// TIA Portal project "Project3" (V15.1)

(* hardware
DEVICE "S71500/ET200MP station_1"  S7-1500 station
   slot 0: "Rail_0"  Rack  6ES7 590-1***0-0AA0
   slot 1: "PLC_1"  CPU 1515-2 PN  6ES7 515-2AM01-0AB0  V2.6
      slot 3: "CPU display_1"  6ES7591-1BA00-0AA0
*)

// ===== PLC "PLC_1"  CPU 1515-2 PN =====

VAR_GLOBAL   // PLC tag table "Default tag table"
   "onss1" AT %M0.0 : Bool;
   "vari" AT %M0.1 : Bool;
   "onss2" AT %M0.2 : Bool;
   "LetIEMPTY" AT %M0.3 : Bool;
   "onss3" AT %M0.4 : Bool;
   "setACTI" AT %M0.5 : Bool;
END_VAR

TYPE "CodeBar"
   STRUCT
      CodeBar : Array[0..8] of Char;
   END_STRUCT;
END_TYPE

DATA_BLOCK "AnalyseCodeBar_DB"   // DB1
{ S7_Optimized_Access := 'TRUE' }
VERSION : 0.1
// stored: InstanceOfName AnalyseCodeBar
"AnalyseCodeBar"
BEGIN
END_DATA_BLOCK

DATA_BLOCK "SysVariables"   // DB2
{ S7_Optimized_Access := 'TRUE' }
VERSION : 0.1
   VAR
      Start : Bool;
      Stop : Bool;
      SysActivated : Bool;
      SysRunning : Bool;
      ActivateSys : Bool;
      usedPPP : Int;
      usedQQ : Int;
      usedD : Int;
      WidgetsQ : Int;
      DoodadsQ : Int;
      WockiesQ : Int;
      CodeBar : String;
      InCodeBar : String;
      AcCodeBar : String;
      PrCodeBar : String;
      onss1 : Bool;
      onss2 : Bool;
      onss3 : Bool;
      onss4 : Bool;
      Oki1 : Bool;
      Oki2 : Bool;
      productType : String;
   END_VAR
BEGIN
END_DATA_BLOCK

DATA_BLOCK "DetectBarCode_DB"   // DB3
{ S7_Optimized_Access := 'TRUE' }
VERSION : 0.1
// stored: InstanceOfName DetectBarCode
"DetectBarCode"
BEGIN
END_DATA_BLOCK

FUNCTION_BLOCK "AnalyseCodeBar"   // FB1, LAD
{ S7_Optimized_Access := 'TRUE' }
VERSION : 0.1
   VAR_INPUT
      ReadedCodeBar : String;
   END_VAR
   VAR_OUTPUT
      PPPportionInt : Int;
      QQportionInt : Int;
      DportionInt : Int;
   END_VAR
   VAR
      PastCodeBar : String;
      ActuelCodeBar : String;
      UsedCodeBar : String;
      ons1 : Bool;
      ons2 : Bool;
      ons3 : Bool;
      ons4 : Bool;
      ons5 : Bool;
      PPPportion : String;
      QQportion : String;
      Dportion : String;
   END_VAR
   VAR_TEMP
      tempPPP : String;
      tempQQ : String;
      tempD : String;
   END_VAR
   VAR_TEMP   // added for the SCL form of the ladder/FBD networks
      _w1 : Bool;
      _w2 : Bool;
   END_VAR
BEGIN

REGION Network 1
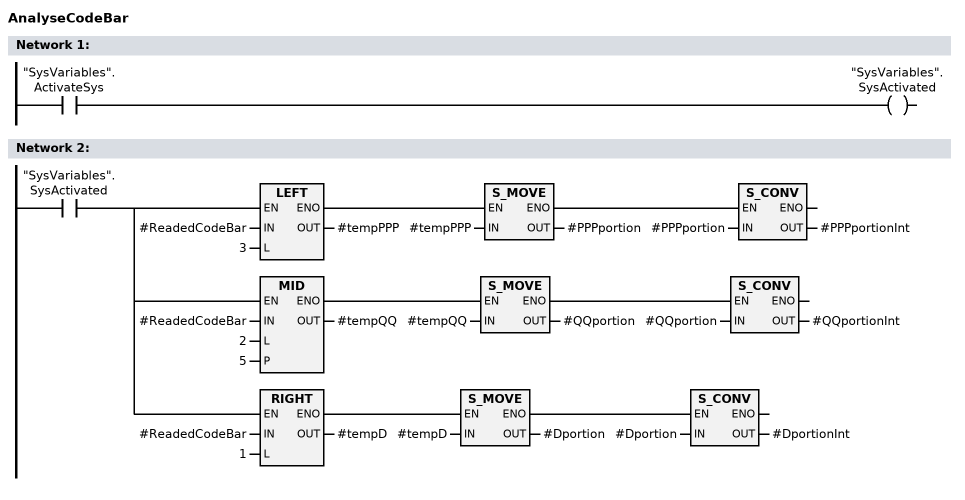
   RUNG wire#powerrail
      Contact( "SysVariables".ActivateSys )
      Coil( "SysVariables".SysActivated )
   END_RUNG
   // the same network as SCL:
   "SysVariables".SysActivated := "SysVariables".ActivateSys;
END_REGION

REGION Network 2
   #_w1 := "SysVariables".SysActivated;
   #_w2 := "SysVariables".SysActivated;
   IF #_w2 THEN
       #tempPPP := LEFT(IN := #ReadedCodeBar, L := 3);
       #PPPportion := #tempPPP;
       #PPPportionInt := S_CONV(IN := #PPPportion);
   END_IF;
   IF #_w1 THEN
       #tempQQ := MID(IN := #ReadedCodeBar, L := 2, P := 5);
       #QQportion := #tempQQ;
       #QQportionInt := S_CONV(IN := #QQportion);
       #tempD := RIGHT(IN := #ReadedCodeBar, L := 1);
       #Dportion := #tempD;
       #DportionInt := S_CONV(IN := #Dportion);
   END_IF;
END_REGION
END_FUNCTION_BLOCK

FUNCTION_BLOCK "DetectBarCode"   // FB2, LAD
{ S7_Optimized_Access := 'TRUE' }
VERSION : 0.1
   VAR_INPUT
      PPPToDetect : Int;
      QQToDetect : Int;
      DToDetect : Int;
   END_VAR
   VAR_OUTPUT
      ProductDirection : String;
      ProductType : String;
      QuanAdded : Int;
      QuanSubded : Int;
   END_VAR
   VAR_IN_OUT
      WidgetsQuan : Int;
      DoodadsQuan : Int;
      WockiesQuan : Int;
   END_VAR
   VAR
      QQPrev : Int;
      QQActuel : Int;
      ons1 : Bool;
      ons2 : Bool;
      ons3 : Bool;
      ons4 : Bool;
      ons5 : Bool;
      ons6 : Bool;
      ons7 : Bool;
      ons8 : Bool;
      ons9 : Bool;
      ons10 : Bool;
      ons11 : Bool;
      ons12 : Bool;
      ons13 : Bool;
      ons14 : Bool;
      ons15 : Bool;
      ons16 : Bool;
      ons17 : Bool;
      ons18 : Bool;
      Tap1 : Bool;
      Tap2 : Bool;
      Tap3 : Bool;
      PPPActuel : Int;
      DActuel : Int;
      PPPPrev : Int;
      DPrev : Int;
      omi1 : Bool;
   END_VAR
   VAR_TEMP
      var1 : Bool;
   END_VAR
   VAR_TEMP   // added for the SCL form of the ladder/FBD networks
      _w1 : Bool;
      _w2 : Bool;
      _w3 : Bool;
      _w4 : Bool;
      _w5 : Bool;
      _w6 : Bool;
      _w7 : Bool;
      _w8 : Bool;
      _w9 : Bool;
      _w10 : Bool;
      _w11 : Bool;
      _w12 : Bool;
      _w13 : Bool;
      _w14 : Bool;
      _w15 : Bool;
      _w16 : Bool;
      _w17 : Bool;
      _w18 : Bool;
   END_VAR
BEGIN

REGION Network 1: PPP to detect
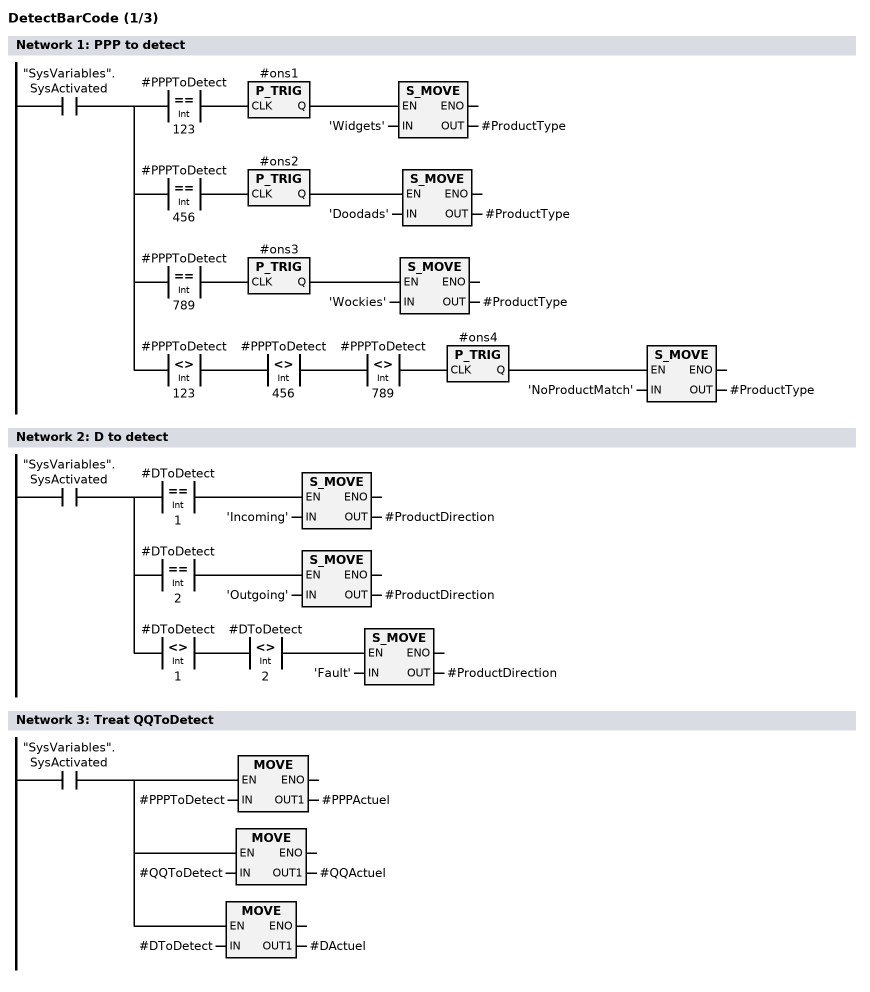
   RUNG wire#powerrail
      Contact( "SysVariables".SysActivated )
      wire#w1
      { S7_Templates := "SrcType := Int" } EQ_Contact(in1 := #PPPToDetect, in2 := 123)
      P_Trig( #ons1 )
      S_Move(in := 'Widgets', out => #ProductType)
   END_RUNG
   RUNG wire#w1
      { S7_Templates := "SrcType := Int" } EQ_Contact(in1 := #PPPToDetect, in2 := 456)
      P_Trig( #ons2 )
      S_Move(in := 'Doodads', out => #ProductType)
   END_RUNG
   RUNG wire#w1
      { S7_Templates := "SrcType := Int" } EQ_Contact(in1 := #PPPToDetect, in2 := 789)
      P_Trig( #ons3 )
      S_Move(in := 'Wockies', out => #ProductType)
   END_RUNG
   RUNG wire#w1
      { S7_Templates := "SrcType := Int" } NE_Contact(in1 := #PPPToDetect, in2 := 123)
      { S7_Templates := "SrcType := Int" } NE_Contact(in1 := #PPPToDetect, in2 := 456)
      { S7_Templates := "SrcType := Int" } NE_Contact(in1 := #PPPToDetect, in2 := 789)
      P_Trig( #ons4 )
      S_Move(in := 'NoProductMatch', out => #ProductType)
   END_RUNG
   // the same network as SCL:
   #_w1 := "SysVariables".SysActivated AND (#PPPToDetect = 123);
   #_w2 := #_w1 AND NOT #ons1;   // rising edge
   #ons1 := #_w1;
   IF #_w2 THEN #ProductType := 'Widgets'; END_IF;
   #_w3 := "SysVariables".SysActivated AND (#PPPToDetect = 456);
   #_w4 := #_w3 AND NOT #ons2;   // rising edge
   #ons2 := #_w3;
   IF #_w4 THEN #ProductType := 'Doodads'; END_IF;
   #_w5 := "SysVariables".SysActivated AND (#PPPToDetect = 789);
   #_w6 := #_w5 AND NOT #ons3;   // rising edge
   #ons3 := #_w5;
   IF #_w6 THEN #ProductType := 'Wockies'; END_IF;
   #_w7 := "SysVariables".SysActivated AND (#PPPToDetect <> 123) AND (#PPPToDetect <> 456) AND (#PPPToDetect <> 789);
   #_w8 := #_w7 AND NOT #ons4;   // rising edge
   #ons4 := #_w7;
   IF #_w8 THEN #ProductType := 'NoProductMatch'; END_IF;
END_REGION

REGION Network 2: D to detect
   RUNG wire#powerrail
      Contact( "SysVariables".SysActivated )
      wire#w1
      { S7_Templates := "SrcType := Int" } EQ_Contact(in1 := #DToDetect, in2 := 1)
      S_Move(in := 'Incoming', out => #ProductDirection)
   END_RUNG
   RUNG wire#w1
      { S7_Templates := "SrcType := Int" } EQ_Contact(in1 := #DToDetect, in2 := 2)
      S_Move(in := 'Outgoing', out => #ProductDirection)
   END_RUNG
   RUNG wire#w1
      { S7_Templates := "SrcType := Int" } NE_Contact(in1 := #DToDetect, in2 := 1)
      { S7_Templates := "SrcType := Int" } NE_Contact(in1 := #DToDetect, in2 := 2)
      S_Move(in := 'Fault', out => #ProductDirection)
   END_RUNG
   // the same network as SCL:
   IF "SysVariables".SysActivated AND (#DToDetect = 1) THEN #ProductDirection := 'Incoming'; END_IF;
   IF "SysVariables".SysActivated AND (#DToDetect = 2) THEN #ProductDirection := 'Outgoing'; END_IF;
   IF "SysVariables".SysActivated AND (#DToDetect <> 1) AND (#DToDetect <> 2) THEN
       #ProductDirection := 'Fault';
   END_IF;
END_REGION

REGION Network 3: Treat QQToDetect
   RUNG wire#powerrail
      Contact( "SysVariables".SysActivated )
      wire#w1
      Move(in := #PPPToDetect, out1 => #PPPActuel)
   END_RUNG
   RUNG wire#w1
      Move(in := #QQToDetect, out1 => #QQActuel)
   END_RUNG
   RUNG wire#w1
      Move(in := #DToDetect, out1 => #DActuel)
   END_RUNG
   // the same network as SCL:
   IF "SysVariables".SysActivated THEN
       #PPPActuel := #PPPToDetect;
       #QQActuel := #QQToDetect;
       #DActuel := #DToDetect;
   END_IF;
END_REGION

REGION Network 4: QQ to detect
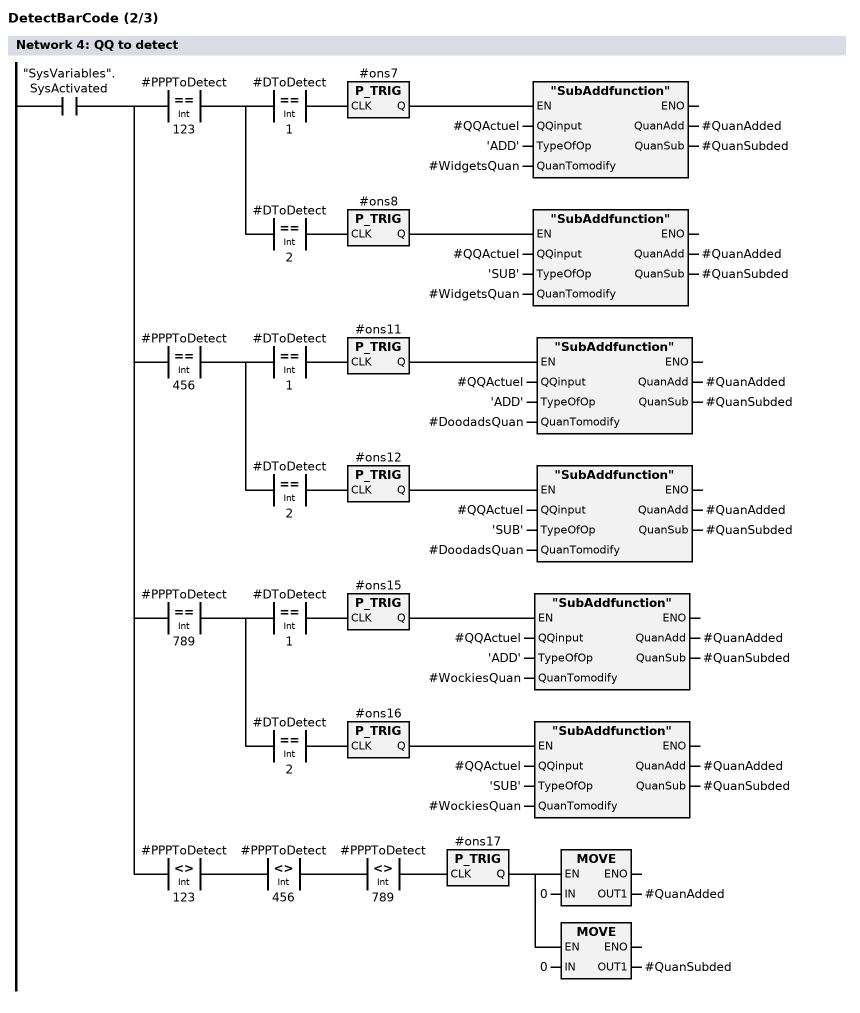
   RUNG wire#powerrail
      Contact( "SysVariables".SysActivated )
      wire#w1
      { S7_Templates := "SrcType := Int" } EQ_Contact(in1 := #PPPToDetect, in2 := 123)
      wire#w2
      { S7_Templates := "SrcType := Int" } EQ_Contact(in1 := #DToDetect, in2 := 1)
      P_Trig( #ons7 )
      "SubAddfunction"(QQinput := #QQActuel, TypeOfOp := 'ADD', QuanTomodify := #WidgetsQuan, QuanAdd => #QuanAdded, QuanSub => #QuanSubded)
   END_RUNG
   RUNG wire#w2
      { S7_Templates := "SrcType := Int" } EQ_Contact(in1 := #DToDetect, in2 := 2)
      P_Trig( #ons8 )
      "SubAddfunction"(QQinput := #QQActuel, TypeOfOp := 'SUB', QuanTomodify := #WidgetsQuan, QuanAdd => #QuanAdded, QuanSub => #QuanSubded)
   END_RUNG
   RUNG wire#w1
      { S7_Templates := "SrcType := Int" } EQ_Contact(in1 := #PPPToDetect, in2 := 456)
      wire#w3
      { S7_Templates := "SrcType := Int" } EQ_Contact(in1 := #DToDetect, in2 := 1)
      P_Trig( #ons11 )
      "SubAddfunction"(QQinput := #QQActuel, TypeOfOp := 'ADD', QuanTomodify := #DoodadsQuan, QuanAdd => #QuanAdded, QuanSub => #QuanSubded)
   END_RUNG
   RUNG wire#w3
      { S7_Templates := "SrcType := Int" } EQ_Contact(in1 := #DToDetect, in2 := 2)
      P_Trig( #ons12 )
      "SubAddfunction"(QQinput := #QQActuel, TypeOfOp := 'SUB', QuanTomodify := #DoodadsQuan, QuanAdd => #QuanAdded, QuanSub => #QuanSubded)
   END_RUNG
   RUNG wire#w1
      { S7_Templates := "SrcType := Int" } EQ_Contact(in1 := #PPPToDetect, in2 := 789)
      wire#w4
      { S7_Templates := "SrcType := Int" } EQ_Contact(in1 := #DToDetect, in2 := 1)
      P_Trig( #ons15 )
      "SubAddfunction"(QQinput := #QQActuel, TypeOfOp := 'ADD', QuanTomodify := #WockiesQuan, QuanAdd => #QuanAdded, QuanSub => #QuanSubded)
   END_RUNG
   RUNG wire#w4
      { S7_Templates := "SrcType := Int" } EQ_Contact(in1 := #DToDetect, in2 := 2)
      P_Trig( #ons16 )
      "SubAddfunction"(QQinput := #QQActuel, TypeOfOp := 'SUB', QuanTomodify := #WockiesQuan, QuanAdd => #QuanAdded, QuanSub => #QuanSubded)
   END_RUNG
   RUNG wire#w1
      { S7_Templates := "SrcType := Int" } NE_Contact(in1 := #PPPToDetect, in2 := 123)
      { S7_Templates := "SrcType := Int" } NE_Contact(in1 := #PPPToDetect, in2 := 456)
      { S7_Templates := "SrcType := Int" } NE_Contact(in1 := #PPPToDetect, in2 := 789)
      P_Trig( #ons17 )
      wire#w5
      Move(in := 0, out1 => #QuanAdded)
   END_RUNG
   RUNG wire#w5
      Move(in := 0, out1 => #QuanSubded)
   END_RUNG
   // the same network as SCL:
   #_w1 := "SysVariables".SysActivated AND (#PPPToDetect = 123);
   #_w2 := #_w1 AND (#DToDetect = 1);
   #_w3 := #_w2 AND NOT #ons7;   // rising edge
   #ons7 := #_w2;
   #_w4 := "SysVariables".SysActivated;
   IF #_w3 THEN
       "SubAddfunction"(QQinput := #QQActuel,
                        TypeOfOp := 'ADD',
                        QuanTomodify := #WidgetsQuan,
                        QuanAdd => #QuanAdded,
                        QuanSub => #QuanSubded);
   END_IF;
   #_w5 := #_w1 AND (#DToDetect = 2);
   #_w6 := #_w5 AND NOT #ons8;   // rising edge
   #ons8 := #_w5;
   IF #_w6 THEN
       "SubAddfunction"(QQinput := #QQActuel,
                        TypeOfOp := 'SUB',
                        QuanTomodify := #WidgetsQuan,
                        QuanAdd => #QuanAdded,
                        QuanSub => #QuanSubded);
   END_IF;
   #_w7 := #_w4 AND (#PPPToDetect = 456);
   #_w8 := #_w7 AND (#DToDetect = 1);
   #_w9 := #_w8 AND NOT #ons11;   // rising edge
   #ons11 := #_w8;
   IF #_w9 THEN
       "SubAddfunction"(QQinput := #QQActuel,
                        TypeOfOp := 'ADD',
                        QuanTomodify := #DoodadsQuan,
                        QuanAdd => #QuanAdded,
                        QuanSub => #QuanSubded);
   END_IF;
   #_w10 := #_w7 AND (#DToDetect = 2);
   #_w11 := #_w10 AND NOT #ons12;   // rising edge
   #ons12 := #_w10;
   IF #_w11 THEN
       "SubAddfunction"(QQinput := #QQActuel,
                        TypeOfOp := 'SUB',
                        QuanTomodify := #DoodadsQuan,
                        QuanAdd => #QuanAdded,
                        QuanSub => #QuanSubded);
   END_IF;
   #_w12 := #_w4 AND (#PPPToDetect = 789);
   #_w13 := #_w12 AND (#DToDetect = 1);
   #_w14 := #_w13 AND NOT #ons15;   // rising edge
   #ons15 := #_w13;
   IF #_w14 THEN
       "SubAddfunction"(QQinput := #QQActuel,
                        TypeOfOp := 'ADD',
                        QuanTomodify := #WockiesQuan,
                        QuanAdd => #QuanAdded,
                        QuanSub => #QuanSubded);
   END_IF;
   #_w15 := #_w12 AND (#DToDetect = 2);
   #_w16 := #_w15 AND NOT #ons16;   // rising edge
   #ons16 := #_w15;
   IF #_w16 THEN
       "SubAddfunction"(QQinput := #QQActuel,
                        TypeOfOp := 'SUB',
                        QuanTomodify := #WockiesQuan,
                        QuanAdd => #QuanAdded,
                        QuanSub => #QuanSubded);
   END_IF;
   #_w17 := #_w4 AND (#PPPToDetect <> 123) AND (#PPPToDetect <> 456) AND (#PPPToDetect <> 789);
   #_w18 := #_w17 AND NOT #ons17;   // rising edge
   #ons17 := #_w17;
   IF #_w18 THEN
       #QuanAdded := 0;
       #QuanSubded := 0;
   END_IF;
END_REGION

REGION Network 5
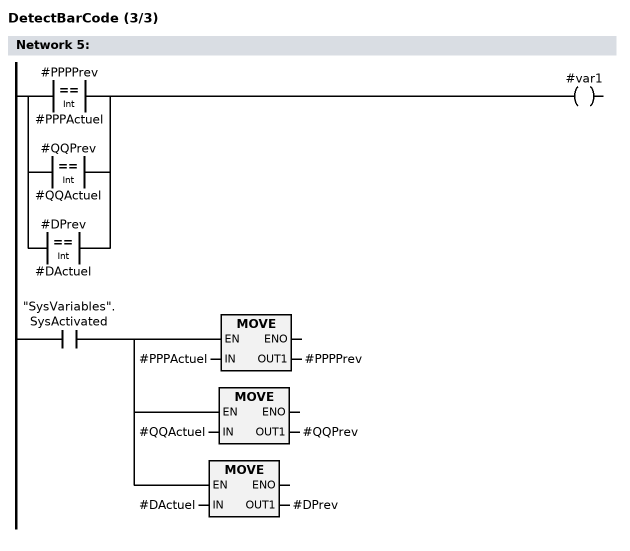
   RUNG wire#powerrail
      { S7_Templates := "SrcType := Int" } EQ_Contact(in1 := #PPPPrev, in2 := #PPPActuel)
      wire#w1
      Coil( #var1 )
   END_RUNG
   RUNG wire#powerrail
      { S7_Templates := "SrcType := Int" } EQ_Contact(in1 := #QQPrev, in2 := #QQActuel)
   END_RUNG wire#w1
   RUNG wire#powerrail
      { S7_Templates := "SrcType := Int" } EQ_Contact(in1 := #DPrev, in2 := #DActuel)
   END_RUNG wire#w1
   RUNG wire#powerrail
      Contact( "SysVariables".SysActivated )
      wire#w2
      Move(in := #PPPActuel, out1 => #PPPPrev)
   END_RUNG
   RUNG wire#w2
      Move(in := #QQActuel, out1 => #QQPrev)
   END_RUNG
   RUNG wire#w2
      Move(in := #DActuel, out1 => #DPrev)
   END_RUNG
   // the same network as SCL:
   #var1 := (#PPPPrev = #PPPActuel) OR (#QQPrev = #QQActuel) OR (#DPrev = #DActuel);
   IF "SysVariables".SysActivated THEN
       #PPPPrev := #PPPActuel;
       #QQPrev := #QQActuel;
       #DPrev := #DActuel;
   END_IF;
END_REGION
END_FUNCTION_BLOCK

FUNCTION "SubAddfunction" : Void   // FC1, LAD
{ S7_Optimized_Access := 'TRUE' }
VERSION : 0.1
   VAR_INPUT
      QQinput : Int;
      TypeOfOp : String;
   END_VAR
   VAR_OUTPUT
      QuanAdd : Int;
      QuanSub : Int;
   END_VAR
   VAR_IN_OUT
      QuanTomodify : Int;
   END_VAR
   VAR_TEMP
      oki1 : Bool;
      oki2 : Bool;
      oki3 : Bool;
   END_VAR
BEGIN

REGION Network 1
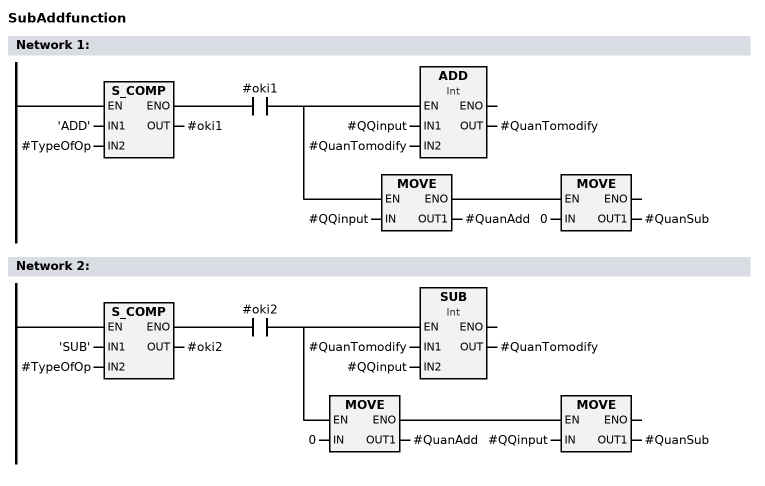
   // ENO of a box is taken as its EN; it also drops when the box reports an error
   S_COMP(IN1 := 'ADD', IN2 := #TypeOfOp, OUT => #oki1);
   IF #oki1 THEN
       #QuanTomodify := #QQinput + #QuanTomodify;
       #QuanAdd := #QQinput;
       #QuanSub := 0;
   END_IF;
END_REGION

REGION Network 2
   // ENO of a box is taken as its EN; it also drops when the box reports an error
   S_COMP(IN1 := 'SUB', IN2 := #TypeOfOp, OUT => #oki2);
   IF #oki2 THEN
       #QuanTomodify := #QuanTomodify - #QQinput;
       #QuanAdd := 0;
       #QuanSub := #QQinput;
   END_IF;
END_REGION
END_FUNCTION

ORGANIZATION_BLOCK "Main"   // OB1, LAD, ProgramCycle
TITLE = "Main Program Sweep (Cycle)"
{ S7_Optimized_Access := 'TRUE' }
VERSION : 0.1
   VAR_INPUT
      Initial_Call : Bool;   // Initial call of this OB
      Remanence : Bool;   // =True, if remanent data are available
   END_VAR
   VAR_TEMP   // added for the SCL form of the ladder/FBD networks
      _w1 : Bool;
   END_VAR
BEGIN

REGION Network 1
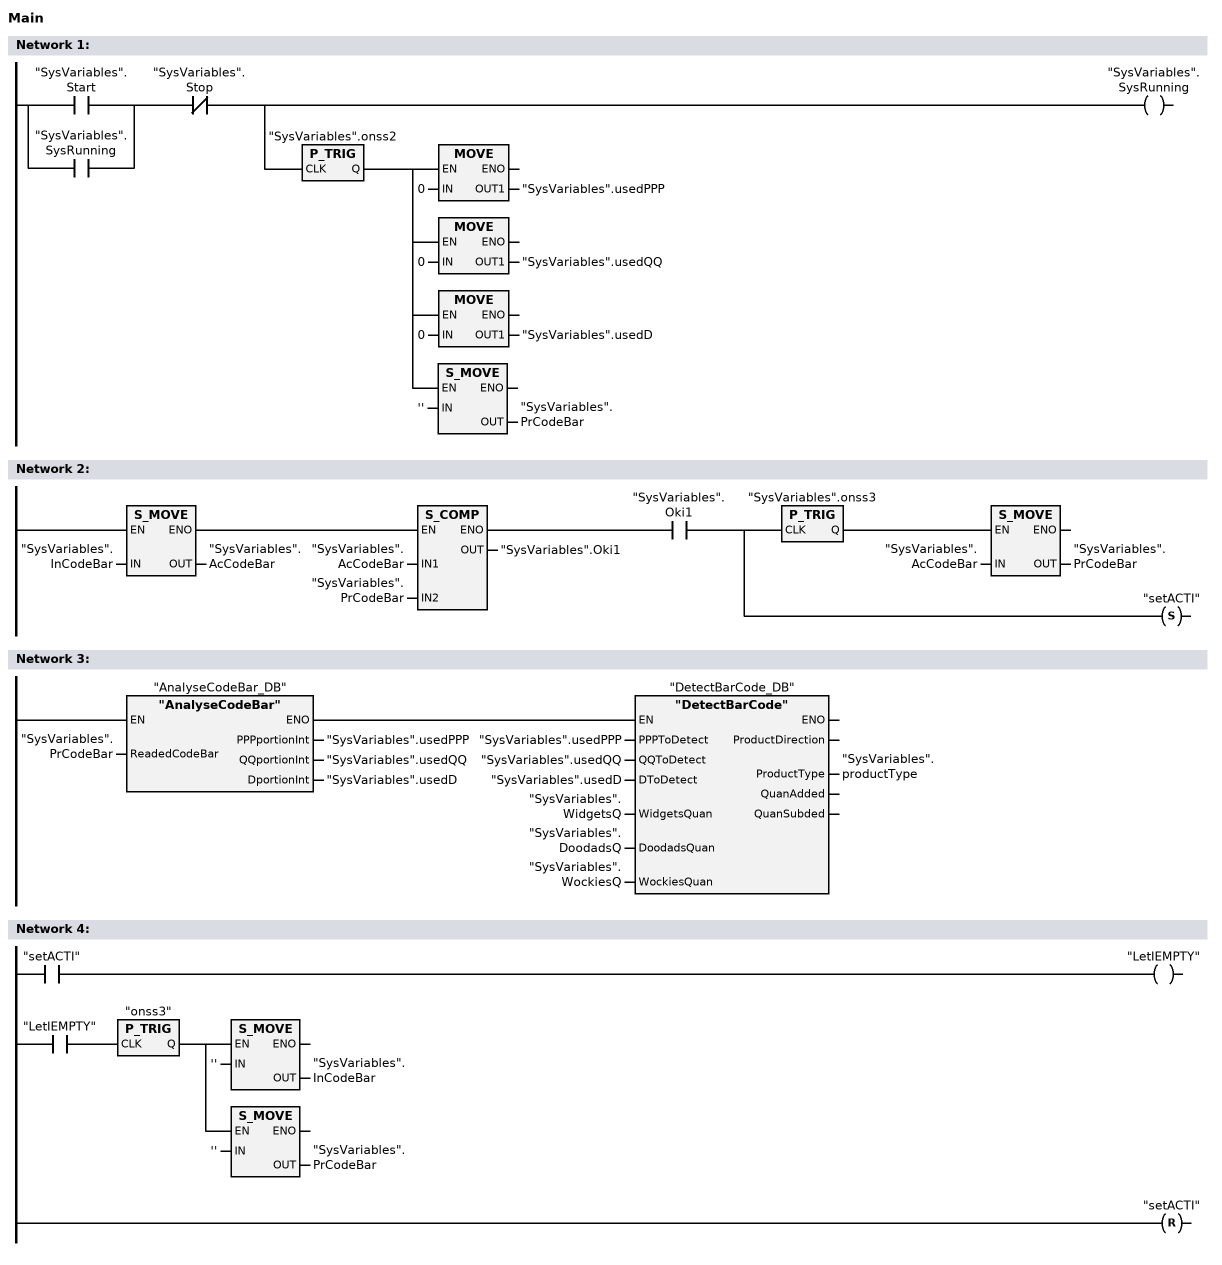
   RUNG wire#powerrail
      Contact( "SysVariables".Start )
      wire#w1
      I_Contact( "SysVariables".Stop )
      wire#w2
      Coil( "SysVariables".SysRunning )
   END_RUNG
   RUNG wire#powerrail
      Contact( "SysVariables".SysRunning )
   END_RUNG wire#w1
   RUNG wire#w2
      P_Trig( "SysVariables".onss2 )
      wire#w3
      Move(in := 0, out1 => "SysVariables".usedPPP)
   END_RUNG
   RUNG wire#w3
      Move(in := 0, out1 => "SysVariables".usedQQ)
   END_RUNG
   RUNG wire#w3
      Move(in := 0, out1 => "SysVariables".usedD)
   END_RUNG
   RUNG wire#w3
      S_Move(in := '', out => "SysVariables".PrCodeBar)
   END_RUNG
   // the same network as SCL:
   "SysVariables".SysRunning := ("SysVariables".Start OR "SysVariables".SysRunning) AND NOT "SysVariables".Stop;
   #_w1 := "SysVariables".SysRunning AND NOT "SysVariables".onss2;   // rising edge
   "SysVariables".onss2 := "SysVariables".SysRunning;
   IF #_w1 THEN
       "SysVariables".usedPPP := 0;
       "SysVariables".usedQQ := 0;
       "SysVariables".usedD := 0;
       "SysVariables".PrCodeBar := '';
   END_IF;
END_REGION

REGION Network 2
   // ENO of a box is taken as its EN; it also drops when the box reports an error
   "SysVariables".AcCodeBar := "SysVariables".InCodeBar;
   S_COMP(IN1 := "SysVariables".AcCodeBar, IN2 := "SysVariables".PrCodeBar, OUT => "SysVariables".Oki1);
   #_w1 := "SysVariables".Oki1 AND NOT "SysVariables".onss3;   // rising edge
   "SysVariables".onss3 := "SysVariables".Oki1;
   IF #_w1 THEN "SysVariables".PrCodeBar := "SysVariables".AcCodeBar; END_IF;
   IF "SysVariables".Oki1 THEN "setACTI" := TRUE; END_IF;
END_REGION

REGION Network 3
   RUNG wire#powerrail
      "AnalyseCodeBar_DB"(ReadedCodeBar := "SysVariables".PrCodeBar, PPPportionInt => "SysVariables".usedPPP, QQportionInt => "SysVariables".usedQQ, DportionInt => "SysVariables".usedD)
      "DetectBarCode_DB"(PPPToDetect := "SysVariables".usedPPP, QQToDetect := "SysVariables".usedQQ, DToDetect := "SysVariables".usedD, WidgetsQuan := "SysVariables".WidgetsQ, DoodadsQuan := "SysVariables".DoodadsQ, WockiesQuan := "SysVariables".WockiesQ, ProductDirection =>, ProductType => "SysVariables".productType, QuanAdded =>, QuanSubded =>)
   END_RUNG
   // the same network as SCL:
   "AnalyseCodeBar_DB"(ReadedCodeBar := "SysVariables".PrCodeBar,   // "AnalyseCodeBar"
                       PPPportionInt => "SysVariables".usedPPP,
                       QQportionInt => "SysVariables".usedQQ,
                       DportionInt => "SysVariables".usedD,
                       ENO => #_w1);
   IF #_w1 THEN
       "DetectBarCode_DB"(PPPToDetect := "SysVariables".usedPPP,   // "DetectBarCode"
                          QQToDetect := "SysVariables".usedQQ,
                          DToDetect := "SysVariables".usedD,
                          WidgetsQuan := "SysVariables".WidgetsQ,
                          DoodadsQuan := "SysVariables".DoodadsQ,
                          WockiesQuan := "SysVariables".WockiesQ,
                          ProductType => "SysVariables".productType);
   END_IF;
END_REGION

REGION Network 4
   RUNG wire#powerrail
      Contact( "setACTI" )
      Coil( "LetIEMPTY" )
   END_RUNG
   RUNG wire#powerrail
      Contact( "LetIEMPTY" )
      P_Trig( "onss3" )
      wire#w1
      S_Move(in := '', out => "SysVariables".InCodeBar)
   END_RUNG
   RUNG wire#w1
      S_Move(in := '', out => "SysVariables".PrCodeBar)
   END_RUNG
   RUNG wire#powerrail
      R_Coil( "setACTI" )
   END_RUNG
   // the same network as SCL:
   "LetIEMPTY" := "setACTI";
   #_w1 := "LetIEMPTY" AND NOT "onss3";   // rising edge
   "onss3" := "LetIEMPTY";
   IF #_w1 THEN
       "SysVariables".InCodeBar := '';
       "SysVariables".PrCodeBar := '';
   END_IF;
   "setACTI" := FALSE;
END_REGION
END_ORGANIZATION_BLOCK